TYPE ST_OutputStationHSOperationalDataGeneral :
STRUCT
	{attribute 'OPC.UA.DA.Description' := 'Dummy (for making struct visible on OPC UA'}
	Dummy						: BOOL;
END_STRUCT
END_TYPE

(* stored: Version 1.1.0.1, ProductVersion 3.1.4024.2
   DUT ST_OutputStationHSOperationalDataGeneral: Id {b253103e-371a-4b67-ba77-ea3323e7b7e4} *)
